// TIA Portal V19 export
VAR_GLOBAL   // PLC tag table "U2EM2_Sr1000"
   errorStatusBits_1_U2Em2 AT %I6017.0 : Bool;
   completionClearControlBits_1_U2Em2 AT %Q6004.0 : Bool;
   latchAndErrorClearControlBits_1_U2Em2 AT %Q6002.0 : Bool;
   handshakeAndGeneralErrorStatusBits_1_U2Em2 AT %I6014.0 : Bool;
   operationInstructionControlBits_1_U2Em2 AT %Q6003.0 : Bool;
   busyStatusBits_1_U2Em2 AT %I6015.0 : Bool;
   unstableReadStatusBits_1_U2Em2 AT %I6019.0 : Bool;
   terminalStatusBits_1_U2Em2 AT %I6018.0 : Bool;
   completionStatusBits_1_U2Em2 AT %I6016.0 : Bool;
   errorStatusByte_1_U2Em2 AT %IB6017 : Byte;
   completionClearControlByte_1_U2Em2 AT %QB6004 : Byte;
   latchAndErrorClearControlByte_1_U2Em2 AT %QB6002 : Byte;
   handshakeAndGeneralErrorStatusByte_1_U2Em2 AT %IB6014 : Byte;
   operationInstructionControlByte_1_U2Em2 AT %QB6003 : Byte;
   busyStatusByte_1_U2Em2 AT %IB6015 : Byte;
   unstableReadStatusByte_1_U2Em2 AT %IB6019 : Byte;
   terminalStatusByte_1_U2Em2 AT %IB6018 : Byte;
   completionStatusByte_1_U2Em2 AT %IB6016 : Byte;
END_VAR
